# EPICS substitutions: EPU60App/Db/globalStatus_sst1.substitutions
file globalStatus.template
{
	# SYS,DEV: All records are prefixed with $(SYS){$(DEV)}
	# CARD: PMAC card num.
	# TMOT: Asyn. communication timeout
	# PORT: PMAC port
	# RING_CHECK_SEVERITY: Alarm level for MACRO Ring Check status. Set to NO_ALARM for MACRO disabled.

	pattern
	{
		CARD, TMOT, PORT, RING_CHECK_SEVERITY
	}
	{
		"0", "4", "PMAC_ETH_PORT", "NO_ALARM"
	}
}
